{attribute 'linkalways'} 
{attribute 'no_explicit_call' := 'This FB is a CLASS and must be accessed using methods or properties'}
{attribute 'enable_dynamic_creation'}
FUNCTION_BLOCK _TcVnArray3_Point2_REAL EXTENDS AliasDatatypeBase
VAR
	localData : TcVnArray3_Point2_REAL;
	activeData : REFERENCE TO TcVnArray3_Point2_REAL REF= localData;
	aliasBaseDatatype : _Array0to2OfTcVnPoint2_REAL;
END_VAR

PROPERTY PUBLIC Address : PVOID
GET
Address := ADR(activeData);
END_GET
END_PROPERTY

METHOD PUBLIC ClearReference
VAR_INPUT
END_VAR
activeData REF= localData;
SetBaseDatatypeReference();
END_METHOD

METHOD PUBLIC Clone : I_Datatype
VAR
    pClone : POINTER TO _TcVnArray3_Point2_REAL;
END_VAR
pClone := __NEW(_TcVnArray3_Point2_REAL);
Clone := pClone^;
END_METHOD

METHOD FB_init : BOOL
VAR_INPUT
	bInitRetains : BOOL; // if TRUE, the retain variables are initialized (warm start / cold start)
	bInCopyCode : BOOL;  // if TRUE, the instance afterwards gets moved into the copy code (online change)
	//InitialValue : TcVnArray4_LREAL; // if possible, not all values can be initialized
END_VAR
//localData := InitialValue; // if possible, not all values can be initialized
SetBaseDatatypeReference();
AddBaseDatatype(aliasBaseDatatype);
END_METHOD

PROPERTY PUBLIC Identifier : T_MAXSTRING
GET
Identifier := 'TcVnArray3_Point2_REAL';
END_GET
END_PROPERTY

METHOD PUBLIC MakeReferenceTo
VAR_INPUT
	ReferenceTarget : REFERENCE TO TcVnArray3_Point2_REAL;
END_VAR
activeData REF= ReferenceTarget;
SetBaseDatatypeReference();
END_METHOD

METHOD PROTECTED SetBaseDatatypeReference
VAR_INPUT
END_VAR
aliasBaseDatatype.MakeReferenceTo(activeData);
END_METHOD

PROPERTY PUBLIC Size : UDINT
GET
Size := SIZEOF(activeData);
END_GET
END_PROPERTY

METHOD TryMakeReferenceTo : BOOL
VAR_INPUT
	Target : I_Datatype;
END_VAR
VAR
	targetAsAlias : I_AliasDatatype;
	pTargetData : POINTER TO TcVnArray3_Point2_REAL;
END_VAR
IF NOT Target.TryResolveAsAliasDatatype(targetAsAlias) THEN
	RETURN;
END_IF

IF targetAsAlias.Identifier <> Identifier THEN
	RETURN;
END_IF

pTargetData := Target.Address;
activeData REF= pTargetData^;
SetBaseDatatypeReference();
TryMakeReferenceTo := TRUE;
END_METHOD

PROPERTY PUBLIC Value : REFERENCE TO TcVnArray3_Point2_REAL
GET
Value REF= activeData;
END_GET
END_PROPERTY

END_FUNCTION_BLOCK

(* stored: Version 1.1.0.1, ProductVersion 3.1.4024.13
   POU _TcVnArray3_Point2_REAL: Id {c200a4d4-20ff-0de0-09e2-4aa7859d2fd3}, SpecialFunc None
   Folder Core: Id {5c5ebd7c-4474-015f-145c-9ae614e90ba6}
   Folder Protected: Id {798f0632-2480-0d6b-337d-9cb7b39fe630}
   Folder Customize: Id {5188a9c5-cd4f-0ad0-05c9-893fdeefc55e}
   Folder Constructor: Id {6c5db715-0ca9-01c0-1747-e67926d31628}
   Property Address: Id {5410cd39-b4bf-054d-3cf9-ef3d1d65bd78}
   Get Get: Id {23a39eb5-a6b1-02ed-3d3a-680eaacb968e}
   Method ClearReference: Id {39dc78be-35af-08b1-08d4-72ef22cda3b7}
   Method Clone: Id {b4e1c370-e8ee-0f33-37dd-77ee5fa47d93}
   Method FB_init: Id {ea84419a-b644-0ea1-2aa5-aac9c662e92f}
   Property Identifier: Id {d866e31e-3d79-0f8f-34a5-0133dd7302f6}
   Get Get: Id {0993ebca-d100-042b-39c2-1cfa1a0a51f3}
   Method MakeReferenceTo: Id {e337bef7-bf4b-0c52-2f1f-719b31b32ec9}
   Method SetBaseDatatypeReference: Id {34477a9b-5a32-010b-22f7-86647bf39faf}
   Property Size: Id {176f352f-8fda-02c7-3b8d-60eca24112ea}
   Get Get: Id {8a3bde55-8cd3-0c28-08ce-a98f3b0d0779}
   Method TryMakeReferenceTo: Id {a3c0fa5d-fd9f-07f9-3afa-04b17d48d7dc}
   Property Value: Id {3fcef3b3-98e2-08da-3a4e-fe2148cef2ce}
   Get Get: Id {84a9fe6d-5ad5-068a-21f9-94085455d9ed} *)
